{attribute 'pack_mode' := '1'}
TYPE ST_ResumePathDataIn :
STRUCT
	iPath						: UINT;			// MM path ID (1-65536)
END_STRUCT
END_TYPE

(* stored: Version 1.1.0.1, ProductVersion 3.1.4024.5
   DUT ST_ResumePathDataIn: Id {9e2ebf1e-0810-4c3e-9688-d8c6e5c59657} *)
